FUNCTION_BLOCK Checkers EXTENDS TcoCore.TcoObject
VAR
    _result : eCheckResult;
END_VAR

METHOD CheckAnalogue : REFERENCE TO Checkers
VAR_INPUT
    Signal : REAL;
END_VAR
VAR_INPUT
    pData : POINTER TO AnalogueValueCheck;
END_VAR
VAR
    _inRange : BOOL;
END_VAR
pData^.Measured := Signal;
_inRange := (Signal >= pData^.Mininum) AND (Signal <= pData^.Maximum);

IF (NOT _inRange AND_THEN _result <= eCheckResult.Passed) THEN
    _result := eCheckResult.Failed;
END_IF;

CheckAnalogue REF= THIS^;
END_METHOD

METHOD HasPassed : BOOL
VAR_INPUT
END_VAR
HasPassed := _result = eCheckResult.Passed;
_result := eCheckResult.None;
END_METHOD

METHOD StartChecks : REFERENCE TO Checkers
VAR_INPUT
END_VAR
_result := eCheckResult.Passed;
StartChecks REF= THIS^;
END_METHOD

END_FUNCTION_BLOCK

(* stored: Version 1.1.0.1, ProductVersion 3.1.4024.9
   POU Checkers: Id {023cac74-18c5-4f8c-9a35-9aaefd8e4a9b}, SpecialFunc None
   Method CheckAnalogue: Id {5d7bbaa0-c7b2-46e6-9f14-895c50556dc3}
   Method HasPassed: Id {ccb7bee4-4b78-4869-a3ed-c3faa2efba11}
   Method StartChecks: Id {2d9a2425-9a31-402b-84f7-4ca5dfabfdf3} *)
